// TIA Portal V21 export
TYPE "Std_Portata"
   STRUCT
      In : Struct
         Impulso : Bool;
      END_STRUCT;
      Prm : Struct
         LitriPerImpulso : Real := 1.0;   // K Correttivo = quanti litri per impulso
         Setpoint_Parziale : Real;
         LitriInVolo : Real;
         UnitàMisura : "Std_UnitàDiMisura";
      END_STRUCT;
      Hmi : Struct
         ResetTotalizzatoreTotale : Bool;   // 1 = Resetta totlizzatore totale
         ResetTotalizzatoreParziale : Bool;   // 1 = Resetta totlizzatore parziale
      END_STRUCT;
      Dati : Struct
         PortataAttuale : Real;
         RimanenteParziale : Real;
         Impulso : Bool;
         TriggerConteggioImpulso : Bool;
         PortataLMin : Real;
         PortataLSec : Real;
         TDurataImpulso : "Std_stTimer";
         MDistanzaImpulsi : Bool;
         FPDistanzaImpulsi : Bool;
      END_STRUCT;
      Allarmi : Struct
         "A" { S7_SetPoint := 'True'} : Array[0.."K_NumAllarmiPerPortate"] of "Std_PrmAllarmeStd";
         WordHMI { S7_SetPoint := 'True'} : Word;
      END_STRUCT;
      Out : Struct
         TotalizzatoreTotaleAttuale : Real;
         TotalizzatoreParzialeAttuale : Real;
         TotalizzatoreParzialeRaggiunto : Bool;
         PortataAttuale : Real;
      END_STRUCT;
   END_STRUCT;
END_TYPE
